NAMESPACE LineB1
FUNCTION_BLOCK FB_Interlock
{ S7_Optimized_Access := 'TRUE' ; Published := 'TRUE' }
VERSION : 0.1

BEGIN
END_FUNCTION_BLOCK
END_NAMESPACE

